FUNCTION_BLOCK "FB_MixingSequencer"
VERSION : 0.1

VAR_INPUT
    // ── Field Instrument Readings ──
    Act_MixTank_Temp    : Real;    // From temperature sensor
    Act_MixTank_Weight  : Real;    // From load cell
    Act_Agitator_RPM    : Real;    // From VFD feedback
    Act_HighShear_RPM   : Real;    // From VFD feedback
    Act_Hopper_Weight   : Real;    // From hopper load cell
    Act_Brix            : Real;    // From Brix sensor (if installed)
    Act_PH              : Real;    // From pH sensor (if installed)
END_VAR

VAR_OUTPUT
    // ── Setpoint Outputs to Field Devices ──
    SP_Agitator_RPM     : Real;    // To agitator VFD
    SP_HighShear_RPM    : Real;    // To high-shear VFD
    SP_Temperature      : Real;    // To heating controller
END_VAR

VAR
    // ── Internal Variables ──
    stepTimer           : TON;     // IEC step timer
    heartbeatTimer      : TON;     // PC watchdog timer
    confirmHoldTimer    : TON;     // Anti-bounce for confirm
    lastHeartbeat       : Bool;    // Previous heartbeat state
    flatStepCounter     : Int;     // Running step count (1-based)
    stepStarted         : Bool;    // Flag: current step outputs have been applied
END_VAR

VAR_TEMP
    iProc               : Int;     // Current process index
    iStep               : Int;     // Current step index
    curStep             : "UDT_ProcessStep";  // Current step data
    stepTimePT          : Time;    // Step time as TIME value
END_VAR

BEGIN

// ═══════════════════════════════════════════════════════
//  1. UPDATE ACTUAL VALUES FROM FIELD
// ═══════════════════════════════════════════════════════
"DB_RecipeData".MixTank_Temp_Act   := Act_MixTank_Temp;
"DB_RecipeData".MixTank_Weight_Act := Act_MixTank_Weight;
"DB_RecipeData".Agitator_RPM_Act   := Act_Agitator_RPM;
"DB_RecipeData".HighShear_RPM_Act  := Act_HighShear_RPM;
"DB_RecipeData".Hopper_Weight_Act  := Act_Hopper_Weight;
"DB_RecipeData".Brix_Act           := Act_Brix;
"DB_RecipeData".PH_Act             := Act_PH;


// ═══════════════════════════════════════════════════════
//  2. PC HEARTBEAT WATCHDOG
// ═══════════════════════════════════════════════════════
IF "DB_RecipeData".PC_Heartbeat <> #lastHeartbeat THEN
    #lastHeartbeat := "DB_RecipeData".PC_Heartbeat;
    #heartbeatTimer(IN := FALSE, PT := T#5s);
END_IF;
#heartbeatTimer(IN := TRUE, PT := T#5s);

IF #heartbeatTimer.Q THEN
    "DB_RecipeData".Error_Code := 1; // PC lost!
END_IF;


// ═══════════════════════════════════════════════════════
//  3. COMMAND HANDLING
// ═══════════════════════════════════════════════════════

// ── START Command ──
// Ensure Recipe isn't loading, is ready, and CRC matches.
IF "DB_RecipeData".StartCmd AND "DB_RecipeData".RecipeReady AND NOT "DB_RecipeData".RecipeLoading THEN

    // Run checksum verify on start if IDLE
    IF "DB_RecipeData".PLC_State = 0 THEN
        "DB_RecipeData".CRC_PLC := "FC_CalcChecksum"();

        IF "DB_RecipeData".CRC_PLC = "DB_RecipeData".CRC_App THEN
            "DB_RecipeData".CRC_Match := TRUE;
            "DB_RecipeData".PLC_State       := 1;
            "DB_RecipeData".Current_Process := 0;
            "DB_RecipeData".Current_Step    := 0;
            "DB_RecipeData".Error_Code      := 0;
            "DB_RecipeData".Batch_Complete  := FALSE;
            #flatStepCounter := 1;
            #stepStarted := FALSE;
        ELSE
            "DB_RecipeData".CRC_Match := FALSE;
            "DB_RecipeData".Error_Code := 4; // CRC Mismatch
        END_IF;
    ELSIF "DB_RecipeData".PLC_State = 3 THEN
        // Resume from pause
        "DB_RecipeData".PLC_State := 1;
    END_IF;

    "DB_RecipeData".StartCmd := FALSE;  // Reset command
END_IF;

// ── PAUSE Command ──
IF "DB_RecipeData".PauseCmd THEN
    IF "DB_RecipeData".PLC_State = 1 OR "DB_RecipeData".PLC_State = 2 THEN
        "DB_RecipeData".PLC_State := 3;  // Paused
    END_IF;
    "DB_RecipeData".PauseCmd := FALSE;
END_IF;

// ── ABORT Command ──
IF "DB_RecipeData".AbortCmd THEN
    "DB_RecipeData".PLC_State       := 0;  // Idle
    "DB_RecipeData".Current_Process := 0;
    "DB_RecipeData".Current_Step    := 0;
    "DB_RecipeData".Step_Done       := FALSE;
    "DB_RecipeData".Batch_Complete  := FALSE;
    #flatStepCounter := 0;
    #stepStarted := FALSE;
    SP_Agitator_RPM  := 0.0;
    SP_HighShear_RPM := 0.0;
    SP_Temperature   := 0.0;
    "DB_RecipeData".AbortCmd := FALSE;
END_IF;


// ═══════════════════════════════════════════════════════
//  4. STEP CONFIRMATION HANDLING (State = 2)
// ═══════════════════════════════════════════════════════
IF "DB_RecipeData".PLC_State = 2 AND "DB_RecipeData".Confirm_Step THEN
    #iProc := "DB_RecipeData".Current_Process;
    #iStep := "DB_RecipeData".Current_Step;

    // Safety: Verify echo
    IF "DB_RecipeData".Confirm_Phase = "DB_RecipeData".Active_Phase
       AND "DB_RecipeData".Confirm_SubStep = "DB_RecipeData".Active_SubStep THEN

        "DB_RecipeData".Step_Done     := FALSE;
        "DB_RecipeData".Confirm_Step  := FALSE;
        #stepStarted := FALSE;

        // Advance
        IF #iStep + 1 < "DB_RecipeData".Processes[#iProc].StepCount AND #iStep < 7 THEN
            "DB_RecipeData".Current_Step := #iStep + 1;
        ELSE
            "DB_RecipeData".Current_Step := 0;
            "DB_RecipeData".Current_Process := #iProc + 1;
        END_IF;

        #flatStepCounter := #flatStepCounter + 1;

        IF "DB_RecipeData".Current_Process >= "DB_RecipeData".ProcessCount THEN
            "DB_RecipeData".PLC_State      := 4;  // DONE
            "DB_RecipeData".Batch_Complete  := TRUE;
            SP_Agitator_RPM  := 0.0;
            SP_HighShear_RPM := 0.0;
            SP_Temperature   := 0.0;
        ELSE
            "DB_RecipeData".PLC_State := 1;  // EXECUTING
        END_IF;
    ELSE
        // Reject
        "DB_RecipeData".Error_Code    := 3;
        "DB_RecipeData".Confirm_Step  := FALSE;
    END_IF;
END_IF;


// ═══════════════════════════════════════════════════════
//  5. MAIN SEQUENCER — EXECUTE (State = 1)
// ═══════════════════════════════════════════════════════
IF "DB_RecipeData".PLC_State = 1 THEN

    #iProc := "DB_RecipeData".Current_Process;
    #iStep := "DB_RecipeData".Current_Step;

    IF #iProc > 31 OR NOT "DB_RecipeData".Processes[#iProc].ProcessActive THEN
        "DB_RecipeData".PLC_State     := 4;
        "DB_RecipeData".Batch_Complete := TRUE;
        SP_Agitator_RPM  := 0.0;
        SP_HighShear_RPM := 0.0;
        SP_Temperature   := 0.0;
        RETURN;
    END_IF;

    #curStep := "DB_RecipeData".Processes[#iProc].Steps[#iStep];

    IF NOT #stepStarted THEN
        SP_Agitator_RPM  := #curStep.AgitatorRPM;
        SP_HighShear_RPM := #curStep.HighShearRPM;
        SP_Temperature   := #curStep.Temperature;
        #stepStarted     := TRUE;

        #stepTimer(IN := FALSE, PT := T#1s);

        "DB_RecipeData".Active_SubStep    := #curStep.StepNo;
        "DB_RecipeData".Active_ActionCode := #curStep.ActionCode;
        "DB_RecipeData".Current_Step_Flat := #flatStepCounter;

        // In real PLC, build string from ProcessNo if needed.
        // e.g., CONCAT('p00', INT_TO_STRING(#curStep.ProcessNo))
    END_IF;

    IF #curStep.IsManual THEN
        "DB_RecipeData".Step_Done  := TRUE;
        "DB_RecipeData".PLC_State  := 2;  // WAIT_CONFIRM
        RETURN;
    END_IF;

    IF #curStep.StepTime > 0 THEN
        #stepTimePT := INT_TO_TIME(#curStep.StepTime * 1000);
        #stepTimer(IN := TRUE, PT := #stepTimePT);

        "DB_RecipeData".Step_Timer_Act := TIME_TO_INT(#stepTimePT - #stepTimer.ET) / 1000;

        IF NOT #stepTimer.Q THEN
            RETURN;
        END_IF;

        #stepTimer(IN := FALSE, PT := #stepTimePT);
    END_IF;

    "DB_RecipeData".Step_Done  := TRUE;
    "DB_RecipeData".PLC_State  := 2;  // WAIT_CONFIRM
    "DB_RecipeData".Step_Timer_Act := 0;

END_IF;

END_FUNCTION_BLOCK
